Fanuc KAREL source: wpspdovrd.kl

PROGRAM wpspdovrd
%NOLOCKGROUP
VAR
  p : POSITION
  q : POSITION
  i : INTEGER
  r : REAL
BEGIN
  WITH $PSPD_OVRD = 100 MOVE TO p
END wpspdovrd
